(* PLC project Unnamed, Unknown Unnamed 1 *)
(* stored: creationDateTime 2020-04-18T01:23:02, modificationDateTime 2020-04-22T00:35:20 *)

PROGRAM mixing_tank
  VAR
    B1 AT %IX100.2 : BOOL;  (* START Button *)
    B2 AT %IX100.3 : BOOL;  (* STOP Button *)
    LS_1 AT %IX100.1 : BOOL;  (* Low-level sensor *)
    LS_2 AT %IX100.0 : BOOL;  (* High-level sensor *)
    V1 AT %QX100.1 : BOOL;  (* Valve 1 actuator *)
    V3 AT %QX100.2 : BOOL;  (* Valve 3 actuator *)
    M AT %QX100.3 : BOOL;  (* Mixer motor actuator *)
  END_VAR
  VAR
    sus : USINT := 0;  (* Internal variable to store pre-pause state *)
    T_5 : TON := 0;  (* Timer *)
    stable : BOOL := 1;  (* Variable to check iterative firing *)
    P1 : BOOL := 1;  (* Init *)
    P2 : BOOL := 0;  (* Filling *)
    P3 : BOOL := 0;  (* Mixing *)
    P4 : BOOL := 0;  (* Draining *)
    P5 : BOOL := 0;  (* Stopped *)
  END_VAR

                        
(* Timer Call *)
T_5(IN:= P3, PT:= T#15000ms);


(* TRANSITIONS *)

  
  (*t1*)
  IF P1 AND NOT P2 AND B1 AND NOT LS_2 THEN
    P1:= 0;
    P2:= 1;
    stable:= 0;
  END_IF;
  
  (*t2*)
  IF P1 AND NOT P3 AND B1 AND LS_2 THEN
    P1:= 0;
    P3:= 1;
    stable:= 0;
  END_IF;
  
  (*t3*)
  IF P2 AND NOT P3 AND LS_2 AND NOT B2 THEN 
    P2:= 0;
    P3:= 1;
    stable:= 0;
  END_IF;
  
  (*t4*)
  IF P3 AND NOT P4 AND T_5.Q AND NOT B2 THEN 
    P3:= 0;
    P4:= 1;
    stable:= 0;
  END_IF;
  
  (*t5*)
  IF P2 AND NOT P5 AND B2 THEN
    P2:= 0;
    P5:= 1;
    sus:= 1;
    stable:= 0;
  END_IF;
  
  (*t6*)
  IF P5 AND NOT P2 AND B1 AND sus=1 THEN 
    P5:= 0;
    P2:= 1;
    stable:= 0;
  END_IF;
  
  (*t7*)
  IF P3 AND NOT P5 AND B2 THEN 
    P3:= 0;
    P5:= 1;
    sus:= 2;
    stable:= 0;
  END_IF;
  
  (*t8*)
  IF P5 AND NOT P3 AND B1 AND sus=2 THEN
    P5:= 0;
    P3:= 1;
    stable:= 0;
  END_IF;
  
  (*t9*)
  IF P4 AND NOT P5 AND B2 THEN
    P4:= 0;
    P5:= 1;
    sus:= 3;
    stable:= 0;
  END_IF;
  
  (*t10*)
  IF P5 AND NOT P4 AND B1 AND sus=3 THEN
    P5:= 0;
    P4:= 1;
    stable:= 0;
  END_IF;
  
  (*t11*)
  IF P4 AND NOT P1 AND NOT LS_1 AND NOT B2 THEN
    P4:= 0;
    P1:= 1;
    stable:= 0;
  END_IF;
  

(* OUTPUTS *)

(*P1/P5*)
IF P1 OR P5 THEN
  V1:= 0;
  V3:= 0;
  M:= 0;
END_IF;

(*P2*)
IF P2 THEN
  V1:= 1;
  V3:= 0;
  M:= 0;
END_IF;

(*P3*)
IF P3 THEN
  V1:= 0;
  V3:= 0;
  M:= 1;
END_IF;

(*P4*)
IF P4 THEN
  V1:= 0;
  V3:= 1;
  M:= 0;
END_IF;









          
END_PROGRAM

CONFIGURATION Config0
  RESOURCE Res0 ON PLC
    TASK task0(INTERVAL := T#20ms, PRIORITY := 0);
    PROGRAM instance0 WITH task0 : mixing_tank;
  END_RESOURCE
END_CONFIGURATION
